TYPE ST_SimulateStage :
STRUCT
	fHighLim	:	LREAL	:=10;
	fLowLim		:	LREAL	:=-10;
	fHighAbs	:	LREAL	:=1;
	fLowAbs		:	LREAL	:=-1;
	absSw		:	BOOL;
END_STRUCT
END_TYPE

(* stored: Version 1.1.0.1, ProductVersion 3.1.4020.12
   DUT ST_SimulateStage: Id {6214c77d-9798-421f-aa02-599b6aa5364b} *)
